(* IEC 61131-3 sources: DemoPumpStation/PumpStation/ports, 4 files *)

(* ---- i_logger.st ---- *)
interface ILogger

    method info
    var_input msg : string; end_var
    end_method

end_interface

(* ---- i_presenter.st ---- *)
interface IPumpStationPresenter

    method buildView : PumpStationViewModel
    var_input controller : ref_to PumpStationController; end_var
    end_method

end_interface

(* ---- i_pump_drive_adapter.st ---- *)
interface IPumpVfdDriveAdapter

    method assignToVfd
    var_input unitId : int; end_var
    end_method

    method transferToBypass
    var_input unitId : int; end_var
    end_method

    method stopUnit
    var_input unitId : int; end_var
    end_method

    method getVfdFrequency : lreal
    end_method

    method getVfdStatus : VfdState
    end_method

end_interface

(* ---- i_scada_modbus.st ---- *)
interface IScadaModbus

method init
	var_input
	    settings_segment : ref_to array [*] of word;
    	feedback_segment : ref_to array [*] of word;
	end_var
end_method

method process_pdi
var_in_out pdi : PumpStationControl; end_var
end_method

method process_pdo
var_input
	ctrl_state : PumpControllerViewModel;
	pumps_state : ref_to array[*] of PumpUnitView;
end_var
end_method

method iterate end_method

end_interface
